// Allocates memory on the heap for a string of defined size.
FUNCTION F_MALLOCSTR : POINTER TO STRING
VAR_INPUT
	Size : T_Size; // Size in bytes
END_VAR

F_MALLOCSTR := __NEW(BYTE, TO_UDINT(Size));

END_FUNCTION

(* stored: Version 1.1.0.1, ProductVersion 3.1.4024.4
   POU F_MALLOCSTR: Id {c3d7e0b0-b075-4883-a6ee-a58ece1984ad}, SpecialFunc None *)
